# EPICS substitutions: ek9000App/Db/EL3162.substitutions
file EL3162.template
{       pattern
        {
                TERMINAL,

        }
        {
        }
}
